FUNCTION_BLOCK ASSEMBLE_AD_FROM_AQ (* this Function combines the 16 AQ (QUARTER) adapters to a AD (DWORD) *)
  (* Standard: 61499-2; Description: Copyright (c) 2026 Meisterschulen am Ostbahnhof SPDX-License-Identifier: EPL-2.0 *)
  (* Version 1.0, 2026-05-16, Franz Höpfinger, Meisterschulen am Ostbahnhof, initial API and implementation and/or initial documentation *)
  PACKAGE adapter::assembling;
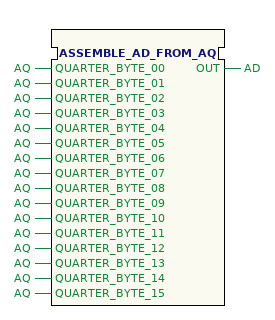
  SOCKETS
    QUARTER_BYTE_00 : adapter::types::unidirectional::AQ; (* Quarter 0 *)
    QUARTER_BYTE_01 : adapter::types::unidirectional::AQ; (* Quarter 1 *)
    QUARTER_BYTE_02 : adapter::types::unidirectional::AQ; (* Quarter 2 *)
    QUARTER_BYTE_03 : adapter::types::unidirectional::AQ; (* Quarter 3 *)
    QUARTER_BYTE_04 : adapter::types::unidirectional::AQ; (* Quarter 4 *)
    QUARTER_BYTE_05 : adapter::types::unidirectional::AQ; (* Quarter 5 *)
    QUARTER_BYTE_06 : adapter::types::unidirectional::AQ; (* Quarter 6 *)
    QUARTER_BYTE_07 : adapter::types::unidirectional::AQ; (* Quarter 7 *)
    QUARTER_BYTE_08 : adapter::types::unidirectional::AQ; (* Quarter 8 *)
    QUARTER_BYTE_09 : adapter::types::unidirectional::AQ; (* Quarter 9 *)
    QUARTER_BYTE_10 : adapter::types::unidirectional::AQ; (* Quarter 10 *)
    QUARTER_BYTE_11 : adapter::types::unidirectional::AQ; (* Quarter 11 *)
    QUARTER_BYTE_12 : adapter::types::unidirectional::AQ; (* Quarter 12 *)
    QUARTER_BYTE_13 : adapter::types::unidirectional::AQ; (* Quarter 13 *)
    QUARTER_BYTE_14 : adapter::types::unidirectional::AQ; (* Quarter 14 *)
    QUARTER_BYTE_15 : adapter::types::unidirectional::AQ; (* Quarter 15 *)
  END_SOCKETS
  PLUGS
    OUT : adapter::types::unidirectional::AD; (* DWORD Output *)
  END_PLUGS
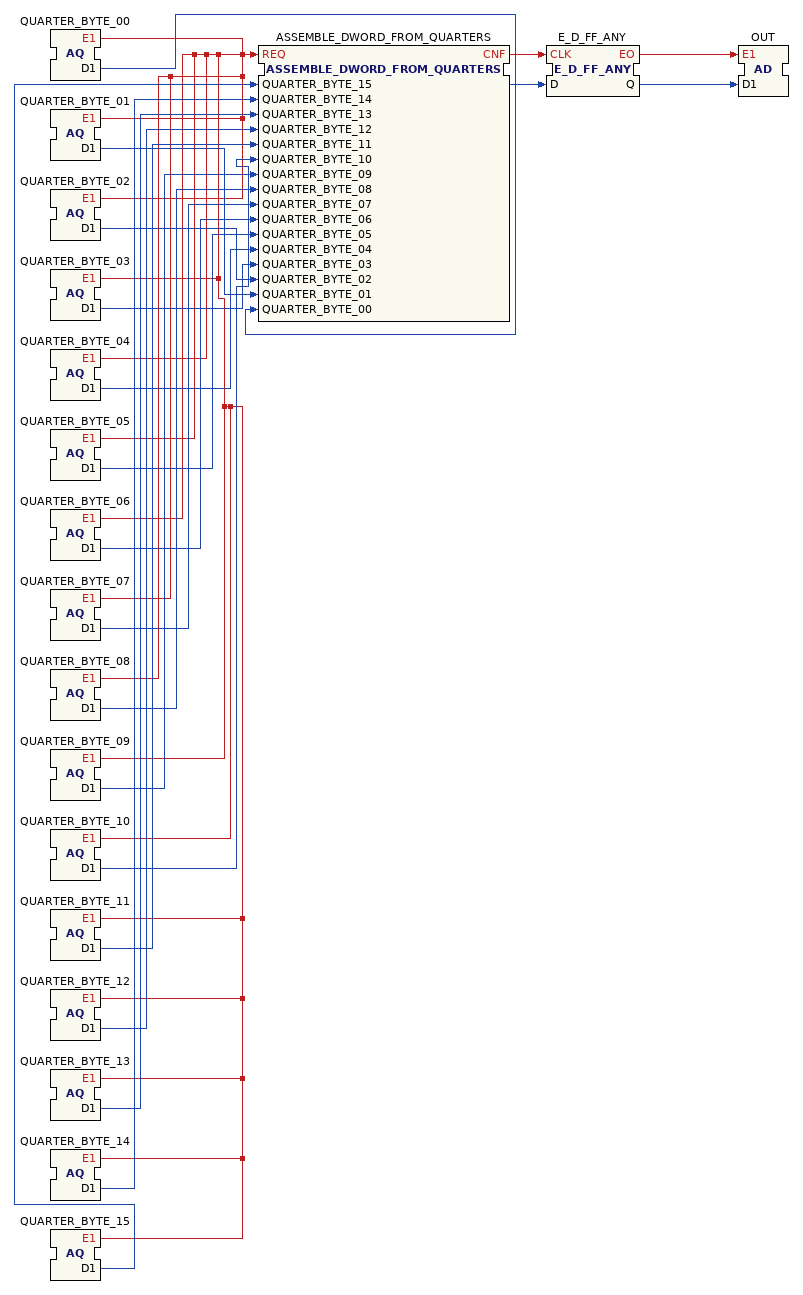
  FBS
    ASSEMBLE_DWORD_FROM_QUARTERS : eclipse4diac::utils::assembling::ASSEMBLE_DWORD_FROM_QUARTERS;
    E_D_FF_ANY : iec61499::events::E_D_FF_ANY;
  END_FBS
  EVENT_CONNECTIONS
    QUARTER_BYTE_00.E1 TO ASSEMBLE_DWORD_FROM_QUARTERS.REQ;
    QUARTER_BYTE_01.E1 TO ASSEMBLE_DWORD_FROM_QUARTERS.REQ;
    QUARTER_BYTE_02.E1 TO ASSEMBLE_DWORD_FROM_QUARTERS.REQ;
    QUARTER_BYTE_03.E1 TO ASSEMBLE_DWORD_FROM_QUARTERS.REQ;
    QUARTER_BYTE_04.E1 TO ASSEMBLE_DWORD_FROM_QUARTERS.REQ;
    QUARTER_BYTE_05.E1 TO ASSEMBLE_DWORD_FROM_QUARTERS.REQ;
    QUARTER_BYTE_06.E1 TO ASSEMBLE_DWORD_FROM_QUARTERS.REQ;
    QUARTER_BYTE_07.E1 TO ASSEMBLE_DWORD_FROM_QUARTERS.REQ;
    QUARTER_BYTE_08.E1 TO ASSEMBLE_DWORD_FROM_QUARTERS.REQ;
    QUARTER_BYTE_09.E1 TO ASSEMBLE_DWORD_FROM_QUARTERS.REQ;
    QUARTER_BYTE_10.E1 TO ASSEMBLE_DWORD_FROM_QUARTERS.REQ;
    QUARTER_BYTE_11.E1 TO ASSEMBLE_DWORD_FROM_QUARTERS.REQ;
    QUARTER_BYTE_12.E1 TO ASSEMBLE_DWORD_FROM_QUARTERS.REQ;
    QUARTER_BYTE_13.E1 TO ASSEMBLE_DWORD_FROM_QUARTERS.REQ;
    QUARTER_BYTE_14.E1 TO ASSEMBLE_DWORD_FROM_QUARTERS.REQ;
    QUARTER_BYTE_15.E1 TO ASSEMBLE_DWORD_FROM_QUARTERS.REQ;
    ASSEMBLE_DWORD_FROM_QUARTERS.CNF TO E_D_FF_ANY.CLK;
    E_D_FF_ANY.EO TO OUT.E1;
  END_CONNECTIONS
  DATA_CONNECTIONS
    ASSEMBLE_DWORD_FROM_QUARTERS. TO E_D_FF_ANY.D;
    E_D_FF_ANY.Q TO OUT.D1;
    QUARTER_BYTE_15.D1 TO ASSEMBLE_DWORD_FROM_QUARTERS.QUARTER_BYTE_15;
    QUARTER_BYTE_14.D1 TO ASSEMBLE_DWORD_FROM_QUARTERS.QUARTER_BYTE_14;
    QUARTER_BYTE_13.D1 TO ASSEMBLE_DWORD_FROM_QUARTERS.QUARTER_BYTE_13;
    QUARTER_BYTE_12.D1 TO ASSEMBLE_DWORD_FROM_QUARTERS.QUARTER_BYTE_12;
    QUARTER_BYTE_11.D1 TO ASSEMBLE_DWORD_FROM_QUARTERS.QUARTER_BYTE_11;
    QUARTER_BYTE_10.D1 TO ASSEMBLE_DWORD_FROM_QUARTERS.QUARTER_BYTE_10;
    QUARTER_BYTE_09.D1 TO ASSEMBLE_DWORD_FROM_QUARTERS.QUARTER_BYTE_09;
    QUARTER_BYTE_08.D1 TO ASSEMBLE_DWORD_FROM_QUARTERS.QUARTER_BYTE_08;
    QUARTER_BYTE_07.D1 TO ASSEMBLE_DWORD_FROM_QUARTERS.QUARTER_BYTE_07;
    QUARTER_BYTE_06.D1 TO ASSEMBLE_DWORD_FROM_QUARTERS.QUARTER_BYTE_06;
    QUARTER_BYTE_05.D1 TO ASSEMBLE_DWORD_FROM_QUARTERS.QUARTER_BYTE_05;
    QUARTER_BYTE_04.D1 TO ASSEMBLE_DWORD_FROM_QUARTERS.QUARTER_BYTE_04;
    QUARTER_BYTE_03.D1 TO ASSEMBLE_DWORD_FROM_QUARTERS.QUARTER_BYTE_03;
    QUARTER_BYTE_02.D1 TO ASSEMBLE_DWORD_FROM_QUARTERS.QUARTER_BYTE_02;
    QUARTER_BYTE_01.D1 TO ASSEMBLE_DWORD_FROM_QUARTERS.QUARTER_BYTE_01;
    QUARTER_BYTE_00.D1 TO ASSEMBLE_DWORD_FROM_QUARTERS.QUARTER_BYTE_00;
  END_CONNECTIONS
END_FUNCTION_BLOCK
